FUNCTION_BLOCK FB_Simplex
VAR
	(* Stored Motor Parameters *)
	bWriteData	: BOOL;

	nTorqueLimit		: INT  := 3; // TorqueLimit for the motor  
	rM_SetPointSpeed	: REAL := 10;		 // Setpoint from user (cmm/s) 
	unControlOption		: UINT := 32;
	
	dnCenterPosition	: DINT;
	dnCCVEndPosition	: DINT := -200000;
	dnCVEndPosition		: DINT := 200000;

	dnPosRegMSB			: DINT;
	dnPosRegLSB			: DINT;
	
	fbModbusRTUMaster 	: MODbusRtuMaster_KL6x22B;
		unVersionNumber		: UINT;
		bMBAddress			: BYTE;
		unQuantity			: UINT; 
		unMBAddr			: UINT;
		unDataLength		: UINT;
		bStartReading		: BOOL;
		unTimeOut			: TIME := T#5S;	
		bBusy				: BOOL;
		bError				: BOOL;
		unErrorID			: UINT;
		unReadBytes			: UINT;
		lnPosition			: LINT;
		SPosition			: DINT;
		nCurr				: INT; // Read register 223	
	stSimplex_SetPosition	: ST_Simplex_SetPosition();	
	stSimplex_Jog			: ST_Simplex_Jog();
	stSimplex_Stop			: ST_Simplex_Stop();
	stSimplex_Reset			: ST_Simplex_Reset();
	stSimplex_Halt			: ST_Simplex_Halt();
	stLoggedValues			: ST_LoggedValues();
	dnRedMSB: BYTE;
END_VAR

(*		fbModbusRTUMaster(	UnitID   := 1,
						  	Quantity := 2,
							MBAddr	 := 200,
							cbLength := 4,
							pMemoryAddr := ADR(lnPosition),
							Execute		:= bWriteData, 
							TimeOut		:= T#5S, 
							Busy		=> bBusy, 
							Error		=> bError,
							ErrorId		=> unErrorID,
							cbRead		=> unReadBytes);		
		fbModbusRTUMaster.ReadRegs();
 *)
 (*
 	fbModbusRTUMaster(	UnitID   := 1,
					  	Quantity := 1,
						MBAddr	 := 449,
						cbLength := 16,
						pMemoryAddr := ADR(dnPosRegMsb),
						Execute		:= bWriteData, 
						TimeOut		:= T#5S, 
						Busy		=> bBusy, 
						Error		=> bError,
						ErrorId		=> unErrorID,
						cbRead		=> unReadBytes);		
	fbModbusRTUMaster.WriteRegs();
*)

{warning 'add method implementation'}
METHOD M_checkNC_settings : BOOL
VAR_INPUT
	//AXIS_REF	: REFERENCE TO Tc2_MC2.AXIS_REF;
END_VAR
END_METHOD

METHOD M_Jog : BOOL
VAR_INPUT
END_VAR
VAR
	bWrite 	: BOOL;	// Write command to Simplex motor
END_VAR
IF stSimplex_Jog.bActive THEN
	stSimplex_Jog.bWriteControlOption := TRUE;
	stSimplex_Jog.bActive := FALSE;
	stSimplex_Jog.bBusy := TRUE;
END_IF

// State to send setpoint velocity to SH200A
IF stSimplex_Jog.bWriteControlOption THEN
	stSimplex_Jog.fbTimerWriteModbus(PT := T#200MS);
	stSimplex_Jog.fbTimerWriteModbus(IN := TRUE);
	IF stSimplex_Jog.fbTimerWriteModbus.Q THEN
		bWrite := TRUE;
		fbModbusRTUMaster(	UnitID   := 1,
						  	Quantity := 1,
							MBAddr	 := 399,
							cbLength := 2,
							pMemoryAddr := ADR(stSimplex_Jog.nControlSetting),
							Execute		:= bWrite, 
							TimeOut		:= T#5S, 
							Busy		=> bBusy, 
							Error		=> bError,
							ErrorId		=> unErrorID,
							cbRead		=> unReadBytes);		
		stSimplex_Jog.bWriteControlOption := FALSE; 
		stSimplex_Jog.bWriteSetPointSpeed := TRUE;
		stSimplex_Jog.fbTimerWriteModbus(IN := FALSE);
	ELSE
		bWrite := FALSE;
		fbModbusRTUMaster(Execute := FALSE);
	END_IF	
	fbModbusRTUMaster.WriteSingleRegister();
	

// State to send control option to SH200A
ELSIF stSimplex_Jog.bWriteSetpointSpeed THEN 
	IF stSimplex_Jog.bSettingsDone THEN
		stSimplex_Jog.bJogForward 			:= TRUE;
		stSimplex_Jog.bSendPosition_LSB 	:= TRUE; 
		stSimplex_Jog.bSendPosition_MSB 	:= TRUE; 
		stSimplex_Jog.bWriteSetPointSpeed 	:= FALSE;
		stSimplex_Jog.bSettingsDone			:= FALSE;
	END_IF
		
	stSimplex_Jog.fbTimerWriteModbus(PT := T#200MS);
	stSimplex_Jog.fbTimerWriteModbus(IN := TRUE);
	stSimplex_Jog.nMaxVelocity := M_MM_TO_SPEED(rMM_SetPoint := rM_SetPointSpeed);
	
	IF stSimplex_Jog.fbTimerWriteModbus.Q THEN
		bWrite := TRUE;
		fbModbusRTUMaster( UnitID   	:= 1,
						   quantity 	:= 1,
						   MBAddr	 	:= 350,
						   cbLength 	:= 2,
						   pMemoryAddr 	:= ADR(stSimplex_Jog.nMaxVelocity),
						   Execute		:= bWrite, 
						   TimeOut		:= T#5S, 
						   Busy			=> bBusy, 
						   Error		=> bError,
						   ErrorId		=> unErrorID,
						   cbRead		=> unReadBytes);	
		stSimplex_Jog.fbTimerWriteModbus(IN := FALSE);
		stSimplex_Jog.bSettingsDone := TRUE;
	ELSE
		bWrite := FALSE;
		fbModbusRTUMaster(Execute := FALSE);
	END_IF
	fbModbusRTUMaster.WriteSingleRegister();
(* STATE 3: JOGGING FORWARD*)
ELSIF stSimplex_Jog.bJogForward THEN
	// Data formatting for Modbus (protcol is broken in the motor)
	dnPosRegMSB := (dnCVEndPosition AND 2#11111111111111110000000000000000);
	dnPosRegLSB := (dnCVEndPosition AND 2#00000000000000001111111111111111);
	
	// If we are done with set-up of new set point read the position for the motor
	IF stSimplex_Jog.bReadPosition THEN
		// Read position from motor
		bWrite := TRUE;
		fbModbusRTUMaster( 	UnitID   	:= 1,
					  		Quantity 	:= 2,
					   		MBAddr	 	:= 200,
					   		cbLength 	:= 4,
					   		pMemoryAddr := ADR(stSimplex_Jog.dnPosition),
					   		Execute		:= bWrite, 
					   		TimeOut		:= T#5S, 
					   		Busy		=> bBusy, 
					   		Error		=> bError,
					   		ErrorId		=> unErrorID,
					   		cbRead		=> unReadBytes);		
		stSimplex_Jog.fbTimerWriteModbus(IN := FALSE);
		fbModbusRTUMaster.ReadRegs();
		IF NOT(bBusy) AND unReadBytes <> 0 THEN
			bWrite := FALSE;
			fbModbusRTUMaster.Execute := FALSE;
		END_IF
	END_IF
	
	IF stSimplex_Jog.bSendPosition_LSB AND stSimplex_Jog.bSendPosition_MSB THEN
		stSimplex_Jog.fbTimerWriteModbus(PT := T#10MS);
		stSimplex_Jog.fbTimerWriteModbus(IN := TRUE);
		
		IF stSimplex_Jog.fbTimerWriteModbus.Q THEN
			fbModbusRTUMaster(	UnitID   := 1,
								Quantity := 1,
								MBAddr	 := 449,
								cbLength := 16,
								pMemoryAddr := ADR(dnPosRegMSB),
								Execute		:= bWrite, 
								TimeOut		:= T#5S, 
								Busy		=> bBusy, 
								Error		=> bError,
								ErrorId		=> unErrorID,
								cbRead		=> unReadBytes);		
			fbModbusRTUMaster.WriteRegs();
			StSimplex_Jog.bSendPosition_MSB := FALSE;
			stSimplex_Jog.fbTimerWriteModbus(IN := FALSE);
		ELSE
			bWrite := FALSE;
			fbModbusRTUMaster(Execute := FALSE);
		END_IF
	ELSIF NOT(stSimplex_Jog.bSendPosition_MSB) AND stSimplex_Jog.bSendPosition_LSB THEN
		stSimplex_Jog.fbTimerWriteModbus(PT := T#10MS);
		stSimplex_Jog.fbTimerWriteModbus(IN := TRUE);
		
		IF stSimplex_Jog.fbTimerWriteModbus.Q THEN
			bWrite := TRUE;
			fbModbusRTUMaster(	UnitID   := 1,
								Quantity := 1,
								MBAddr	 := 450,
								cbLength := 16,
								pMemoryAddr := ADR(dnPosRegLSB),
								Execute		:= bWrite, 
								TimeOut		:= T#5S, 
								Busy		=> bBusy, 
								Error		=> bError,
								ErrorId		=> unErrorID,
								cbRead		=> unReadBytes);		
			fbModbusRTUMaster.WriteRegs();
			StSimplex_Jog.bSendPosition_LSB := FALSE;	
			stSimplex_Jog.fbTimerWriteModbus(IN := FALSE);
		ELSE
			bWrite := FALSE;
			fbModbusRTUMaster(Execute := FALSE);
		END_IF
	ELSIF NOT(stSimplex_Jog.bSendPosition_MSB) AND NOT(stSimplex_Jog.bSendPosition_LSB) THEN
		fbModbusRTUMaster.WriteRegs();
		stSimplex_Jog.bReadPosition := TRUE;
	END_IF		

	IF stSimplex_Jog.dnPosition >= dnCVEndPosition THEN
		stSimplex_Jog.bJogForward		:= FALSE;
		stSimplex_Jog.bJogBackwards 	:= TRUE;
		stSimplex_Jog.bReadPosition 	:= FALSE;
		stSimplex_Jog.bSendPosition_LSB := TRUE;
		stSimplex_Jog.bSendPosition_MSB := TRUE;
		fbModbusRTUMaster.Execute 		:= FALSE;
	END_IF

(* STATE 4: JOGGING BACKWARDS*)
ELSIF stSimplex_Jog.bJogBackwards THEN
	dnPosRegMSB := (dnCCVEndPosition AND 2#11111111111111110000000000000000);
	dnPosRegLSB := (dnCCVEndPosition AND 2#00000000000000001111111111111111);
	
	// Read the position of the motor (True if we are done with the set-up)
	IF stSimplex_Jog.bReadPosition THEN
		// Read position from motor
		bWrite := TRUE;
		fbModbusRTUMaster( 	UnitID   	:= 1,
					  		Quantity 	:= 2,
					   		MBAddr	 	:= 200,
					   		cbLength 	:= 4,
					   		pMemoryAddr := ADR(stSimplex_Jog.dnPosition),
					   		Execute		:= bWrite, 
					   		TimeOut		:= T#5S, 
					   		Busy		=> bBusy, 
					   		Error		=> bError,
					   		ErrorId		=> unErrorID,
					   		cbRead		=> unReadBytes);		
		fbModbusRTUMaster.ReadRegs();
		IF NOT(bBusy) AND unReadBytes <> 0 THEN
			bWrite := FALSE;
			fbModbusRTUMaster.Execute := FALSE;
		END_IF
	END_IF		
	
	IF stSimplex_Jog.bSendPosition_LSB AND stSimplex_Jog.bSendPosition_MSB THEN
		stSimplex_Jog.fbTimerWriteModbus(PT := T#10MS);
		stSimplex_Jog.fbTimerWriteModbus(IN := TRUE);
		
		IF stSimplex_Jog.fbTimerWriteModbus.Q THEN
			fbModbusRTUMaster(	UnitID   := 1,
								Quantity := 1,
								MBAddr	 := 449,
								cbLength := 16,
								pMemoryAddr := ADR(dnPosRegMSB),
								Execute		:= bWrite, 
								TimeOut		:= T#5S, 
								Busy		=> bBusy, 
								Error		=> bError,
								ErrorId		=> unErrorID,
								cbRead		=> unReadBytes);
			stSimplex_Jog.fbTimerWriteModbus(IN := FALSE);
			fbModbusRTUMaster.WriteRegs();
			StSimplex_Jog.bSendPosition_MSB := FALSE;
		ELSE
			bWrite := FALSE;
			fbModbusRTUMaster(Execute := FALSE);
		END_IF
	ELSIF NOT(stSimplex_Jog.bSendPosition_MSB) AND stSimplex_Jog.bSendPosition_LSB THEN	
		stSimplex_Jog.fbTimerWriteModbus(PT := T#10MS);
		stSimplex_Jog.fbTimerWriteModbus(IN := TRUE);
		
		IF stSimplex_Jog.fbTimerWriteModbus.Q THEN
			bWrite := TRUE;
			fbModbusRTUMaster(	UnitID   := 1,
								Quantity := 1,
								MBAddr	 := 450,
								cbLength := 16,
								pMemoryAddr := ADR(dnPosRegLSB),
								Execute		:= bWrite, 
								TimeOut		:= T#5S, 
								Busy		=> bBusy, 
								Error		=> bError,
								ErrorId		=> unErrorID,
								cbRead		=> unReadBytes);
			stSimplex_Jog.fbTimerWriteModbus(IN := FALSE);		
			fbModbusRTUMaster.WriteRegs();
			StSimplex_Jog.bSendPosition_LSB := FALSE;	
		ELSE
			bWrite := FALSE;
			fbModbusRTUMaster(Execute := FALSE);
		END_IF
	ELSIF NOT(stSimplex_Jog.bSendPosition_MSB) AND NOT(stSimplex_Jog.bSendPosition_LSB) THEN
		fbModbusRTUMaster.WriteRegs();
		stSimplex_Jog.bReadPosition := TRUE;
	END_IF
	
	IF stSimplex_Jog.dnPosition >= dnCCVEndPosition THEN
		stSimplex_Jog.bJogForward		:= TRUE;
		stSimplex_Jog.bJogBackwards 	:= FALSE;
		stSimplex_Jog.bReadPosition 	:= FALSE;
		stSimplex_Jog.bSendPosition_LSB := TRUE;
		stSimplex_Jog.bSendPosition_MSB := TRUE;
		fbModbusRTUMaster.Execute 		:= FALSE;
	END_IF	
END_IF

IF stSimplex_Jog.bDone OR stSimplex_Jog.bCommandAborted THEN
	stSimplex_Jog.bJogForward			:= FALSE;
	stSimplex_Jog.bJogBackwards 		:= FALSE;
	stSimplex_Jog.bWriteSetpointSpeed 	:= FALSE;
	stSimplex_Jog.bWriteControlOption 	:= FALSE;
	stSimplex_Jog.bBusy   				:= FALSE;
	stSimplex_Jog.bActive 				:= FALSE;
END_IF
END_METHOD

METHOD M_LogValues : BOOL
VAR_INPUT
	//AXIS_REF	: REFERENCE TO Tc2_MC2.AXIS_REF;
END_VAR
VAR
	nValue : INT;
	nReadBytes : UINT;
END_VAR
(*
IF NOT(bBusy) THEN
	fbModbusRTUMaster(	UnitID   := 1,
					  	Quantity := 1,
						MBAddr	 := 208,
						cbLength := 2,
						pMemoryAddr := ADR(nValue),
						Execute		:= TRUE, 
						TimeOut		:= T#5S, 
						Busy		=> bBusy, 
						Error		=> bError,
						ErrorId		=> unErrorID,
						cbRead		=> nReadBytes);		
	fbModbusRTUMaster.WriteSingleRegister();
END_IF
IF nReadBytes <> 0 THEN
	stLoggedValues.nMotorFluxVoltage := nValue;
END_IF
*)
// Typiskt är 50/200 mm per varv = 0.25 mm per varv 

// 400, uint, värde 32 är speed control för position (Håll en viss fart till position är uppnått) 




// 340, int, unit is positions per second / 16, 0..25600
END_METHOD

METHOD M_MM_TO_SPEED : INT;
VAR_INPUT
	rMM_SetPoint : REAL; 
END_VAR
M_MM_TO_SPEED := REAL_TO_INT(rMM_Setpoint*256*0.25);
END_METHOD

{warning 'add method implementation'}
METHOD M_ResetDrive : BOOL
VAR_INPUT
	//AXIS_REF	: REFERENCE TO Tc2_MC2.AXIS_REF;
END_VAR
END_METHOD

{warning 'add method implementation'}
METHOD M_SetPositionOffset : BOOL
VAR_INPUT
	//AXIS_REF	: REFERENCE TO Tc2_MC2.AXIS_REF;
END_VAR
VAR
	//stMC_SetPosition : ST_MC_SetPosition;
END_VAR
VAR CONSTANT
	// Variables for calculation of the speed
END_VAR
//stMC_Setposition.bExecute := TRUE;
END_METHOD

METHOD M_SetSpeed : BOOL
VAR_INPUT
	//AXIS_REF	: REFERENCE TO Tc2_MC2.AXIS_REF;
END_VAR
VAR
	bState1 	: BOOL; // Write setpoint
	bState2		: BOOL; // Start moving 
	bState3		: BOOL; // Error or end position reach 
END_VAR
// Typiskt är 50/200 mm per varv = 0.25 mm per varv 

// 400, uint, värde 32 är speed control för position (Håll en viss fart till position är uppnått) 




// 340, int, unit is positions per second / 16, 0..25600
END_METHOD

{warning 'add method implementation'}
METHOD M_SetTorqueLimit : BOOL
VAR_INPUT
	//AXIS_REF	: REFERENCE TO Tc2_MC2.AXIS_REF;
END_VAR
VAR_OUTPUT
	bQued	: BOOL;	
END_VAR
VAR
	bBusy 		: BOOL;
	bExecute	: BOOL;
	bError		: BOOL;
	unErrorID	: UINT; 
	nReadBytes	: UINT;
END_VAR
(*// Write register 203!! 
fbModbusRTUMaster(	UnitID   := 1,
				  	Quantity := 1,
					MBAddr	 := 204,
					cbLength := 1,
					pMemoryAddr := ADR(nTorqueLimit),
					Execute		:= TRUE, 
					TimeOut		:= T#5S, 
					Busy		=> bBusy, 
					Error		=> bError,
					ErrorId		=> unErrorID,
					cbRead		=> nReadBytes);
				

IF NOT(bBusy) THEN
	fbModbusRTUMaster.WriteSingleRegister();
	bQued	:= FALSE;
ELSE
	bQued	:= TRUE;
END_IF
*)
END_METHOD

METHOD M_SetZeroRef : BOOL
VAR_INPUT
END_VAR
END_METHOD

END_FUNCTION_BLOCK

(* stored: Version 1.1.0.1, ProductVersion 3.1.4020.12
   POU FB_Simplex: Id {668ab83c-799c-4a0b-96ba-50b562212dee}, SpecialFunc None
   Folder Scaling: Id {1d439a6b-5024-48bb-868f-a4701606a7fd}
   Method M_checkNC_settings: Id {cfbd57d8-d8ed-43d8-a0a0-ea06701a4dc3}
   Method M_Jog: Id {79f88ce3-dc88-4de6-919b-8d632ea73062}
   Method M_LogValues: Id {29f4707f-0732-49c7-9c02-bbb745d728e4}
   Method M_MM_TO_SPEED: Id {25a2b7af-bf4e-4298-978e-f415ad9bce76}
   Method M_ResetDrive: Id {f639bab4-0de1-4dd6-8ddf-997fbfefdbe5}
   Method M_SetPositionOffset: Id {8d951990-4f16-45c3-85b6-58c87d8d0b97}
   Method M_SetSpeed: Id {2d9fd325-2eed-4646-ad15-d3444a3ac3e2}
   Method M_SetTorqueLimit: Id {dd7800fe-2de1-43a4-a1b9-9af2c8ecf0d5}
   Method M_SetZeroRef: Id {86ea4837-fbd4-4612-ad57-497cb308b485} *)
